// SIMATIC S7-200 project (STEP 7-Micro/WIN), CPU 221 REL 01.10

ORGANIZATION_BLOCK 主程序:OB1
TITLE=程序注释
BEGIN
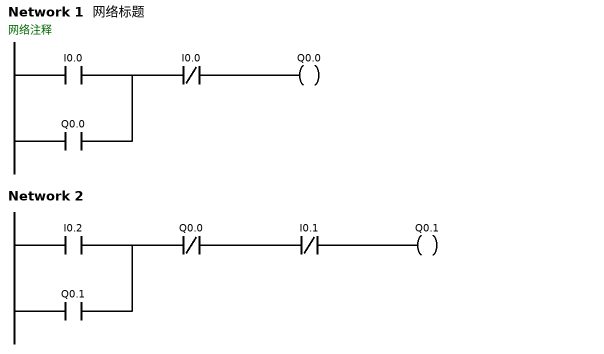
Network 1 // 网络标题
// 网络注释
LD     I0.0
O      Q0.0
AN     I0.0
=      Q0.0
Network 2
LD     I0.2
O      Q0.1
AN     Q0.0
AN     I0.1
=      Q0.1
END_ORGANIZATION_BLOCK
